FUNCTION_BLOCK SU2 (* Basic FB with empty ECC *)
  (* Standard: 61499-2 *)
  (* Version 1.0, 2025-03-31, 06220625900 *)
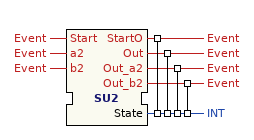
  EVENT_INPUT
    Start;
    a2;
    b2;
  END_EVENT
  EVENT_OUTPUT
    StartO WITH State;
    Out WITH State;
    Out_a2 WITH State;
    Out_b2 WITH State;
  END_EVENT
  VAR_OUTPUT
    State : INT := 1;
  END_VAR
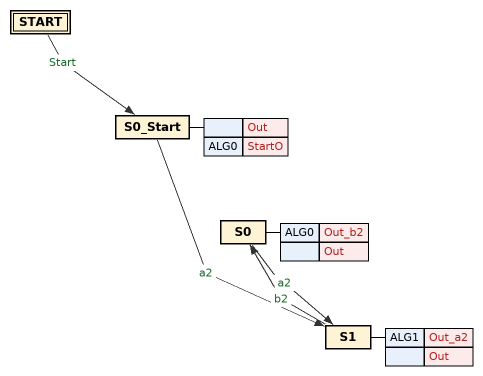
  EC_STATES
    START; (* Initial State *)
    S0_Start : -> Out, ALG0 -> StartO;
    S0 : ALG0 -> Out_b2, -> Out;
    S1 : ALG1 -> Out_a2, -> Out;
  END_STATES
  EC_TRANSITIONS
    START TO S0_Start := Start;
    S0_Start TO S1 := a2;
    S0 TO S1 := a2;
    S1 TO S0 := b2;
  END_TRANSITIONS
  ALGORITHM ALG0 IN ST:
State:=0;
  END_ALGORITHM
  ALGORITHM ALG1 IN ST:
State:=1;
  END_ALGORITHM
END_FUNCTION_BLOCK
